// TIA Portal V20 export
DATA_BLOCK "instRfidMobile"   // DB283
// stored: InstanceOfName LER_RFID_Mobile, InstanceOfType FB
"LER_RFID_Mobile"
   // VAR_INPUT
   //    enable : Bool;
   //    enableManualCmds : Bool;
   // END_VAR
   // VAR_OUTPUT
   //    error : Bool;
   //    status : DWord;
   // END_VAR
   // VAR_IN_OUT
   //    IdentRfAntena : "LSicar_typeIdentInterfaceHmi";
   //    moduleInterface : "LER_typeMobileRFIDInterface";
   // END_VAR
   // VAR
   //    instTRCV_C : TRCV_C;
   //    statConnectionData : TCON_IP_v4;
   //    statTrcvUDT : "LER_typeTrcvUDT";
   //    statResultRFIDReset : Bool;
   //    statPulse : Array[0..9] of Bool;
   //    statTonTimer : TON_TIME;
   //    statBobinData : IID_IN_I_81;
   //    statRFID_str : String[32];
   //    statEPCID_str : String[32];
   //    statHi : Byte;
   //    statLo : Byte;
   //    statHexArray : Array[0..15] of Char;
   // END_VAR
BEGIN
END_DATA_BLOCK
